FUNCTION_BLOCK FB_ModbusReadCoils
////////////////// 
// Read Modbus TCP/IP on Rising Edge of Trigger ClockRead. Returns alarm and stop modbus Read after three consecutive Modbus attempts that failed. 
//////////////////

VAR_INPUT
	
	// Modbus ReadRegs FB inputs
	pDestAddr 	: POINTER TO BYTE ; // Pointer to variable in which the read data have to be stored
	sIPAddr 	: STRING(15);		// Modbus server device IP adress
	tTimeout 	: TIME;				// Timeout
	nTcpPort 	: UINT;
	nQuantity 	: WORD;				// Quantity of words to be read
	nMBAddr 	: WORD ;			// Starting Register adress
	
	cbLength 	: UDINT;			// Length of variable to host the read data
	nUnitID 	: BYTE;				// Unit ID in case of serial connexion after modbus server. Usually equals to 1
	
	ClockRead	: BOOL; 			// Rising Edge Modbus Trigger
	Reset		: BOOL; 			// Reset Trigger to clean alarm and counter.
	
END_VAR

VAR_OUTPUT
	ErrorId			: UDINT;	// Error Id returned by FB ( see ADS error Code ) . 
	
	Busy			: BOOL ;	// FB busy to proceed command
	ModbusReadAlarm	: BOOL; 	// Alarm if three modbus attempt failed.
	OUT_NbRead		: UDINT;
END_VAR

VAR
	R_TRIG 				: R_TRIG; 			// Rising edge detection for the trigger.
	FB_MBReadCoils 		: FB_MBReadCoils; 	// Multiple registers reading
	
	Step				: INT; 				// Grafcet step
	AlarmCounter		: INT; 				// Alarm Counter. Incremennted if modbus errOR  Alarm if counter =3 , resetable.  

	
END_VAR

// ALARM MANAGEMENT //

	IF AlarmCounter=3 THEN 
		ModbusReadAlarm 	:=TRUE;
		
	ELSE
		ModbusReadAlarm := FALSE;
		ErrorId			:= 0;
		
	END_IF


// MODBUS SEQUENCE //
CASE Step OF 
	0:
		R_TRIG(CLK :=ClockRead);
		
		IF R_TRIG.Q THEN 
			Step :=1;
			Busy := TRUE;
			OUT_NbRead := 0;
		END_IF
	1:
	   FB_MBReadCoils(
	  			sIPAddr:= sIPAddr , 
				nTCPPort:= nTcpPort ,
				nUnitID:= nUnitID,
				nQuantity:= nQuantity,
				nMBAddr:= nMBAddr, 
				cbLength:= cbLength, 
				pDestAddr:= pDestAddr, 
				bExecute:= TRUE,
				tTimeout:= tTimeout,
				cbRead => OUT_NbRead
				);
				
		IF NOT FB_MBReadCoils.bBusy AND NOT FB_MBReadCoils.bError THEN
			FB_MBReadCoils(bExecute:= FALSE);
			AlarmCounter	:=0; // Reset counter after successful modbus read. 
			Step 			:=0;
			Busy := FALSE;
		ELSIF NOT FB_MBReadCoils.bBusy AND FB_MBReadCoils.bError THEN
			FB_MBReadCoils(bExecute:= FALSE);
			AlarmCounter 	:= MIN(AlarmCounter+1,3) ; 
			ErrorId			 :=FB_MBReadCoils.nErrId;
			Step 			:=0;
			Busy := FALSE;
		END_IF
		
END_CASE

// RESET //
	IF Reset THEN 
			AlarmCounter 		:= 0 ; 
			ErrorId 			:= 0 ; 
			ModbusReadAlarm 	:=FALSE;
			Reset 				:= FALSE;
			FB_MBReadCoils		(bExecute := FALSE);
	END_IF

// BUSY //

END_FUNCTION_BLOCK

(* stored: Version 1.1.0.1, ProductVersion 3.1.4024.6
   POU FB_ModbusReadCoils: Id {1b435c3e-f7f4-430d-ba92-14b579f9eca6}, SpecialFunc None *)
